Universal Robots PolyScope program: example2.urp

ProgramRoot directory=/home/ur/ursim-3.1/programs; kinematics=(a=[0, -0.425, -0.39225, 0, 0, 0], d=[0.08916, 0, 0, 0.10915, 0.09465, 0.0823], alpha=[1.5708, 0, 0, 1.5708, -1.5708, 0], deltaTheta=[0, 0, 0, 0, 0, 0], status=notInitialized); lastSavedInVersion=(project__name=Polyscope, major__version=3, minor__version=1, svn__revision=17779, build__date=Jun 04 2015, 18:29:53); name=example2; programVersion=(project__name=Polyscope, major__version=3, minor__version=1, svn__revision=17779, build__date=Jun 04 2015, 18:29:53); robotEnvironmentFileName=default; serialNumberRobot=2015350001
  BeforeStart description=COMMAND_SEQUENCE_BEFORE_PROGRAM_START; name=BeforeStart
    Script type=1; cachedFileContents=def getBitValueFromInt(intVal, bitNumber):
      |   a = 1
      |   i = 1
      |   while (i < bitNumber) :
      |     i=i+1
      |     a = a * 2
      |   end
      |   b = floor(intVal / a)
      |   return ((b/2) != floor(b/2))
      | end
      | 
      | def getIntWithBitSet(originalIntVal, bitNumber, bitValue) :
      |   a = 1
      |   i = 1
      |   while (i < bitNumber) :
      |     i=i+1
      |     a = a * 2
      |   end
      |   b = floor(originalIntVal / a)
      |   c = originalIntVal
      |   if ((b/2) == floor(b/2)) :
      |     if (bitValue == True) :
      |       c = c + a
      |     end
      |   else :
      |     if (bitValue == False) :
      |       c = c - a
      |     end
      |   end
      |   return c
      | end; scriptFile=/home/ur/ursim-3.1/programs/Bit_Functions.script
  MainProgram cartesianAcceleration=1.2; cartesianSpeed=0.25; jointAcceleration=1.3962634015954636; jointSpeed=1.0471975511965976; sharedProcessMoveBlendRadius=0.025; motionType=JOINT_SPACE; runOnlyOneCycle=true
    Assignment expr=1000; operatorValueType=INTEGER; valueSource=EXPRESSION
    Assignment expr=getIntWithBitSet(ExpressionVariableNode,2, True ); operatorValueType=INTEGER; valueSource=EXPRESSION
